FUNCTION_BLOCK Master_Axis
VAR_INPUT
	(*Linked_Axis		: AXIS_REF;*)
END_VAR
VAR_OUTPUT
END_VAR
VAR
	Linked_Axis		: AXIS_REF;
	// Motion Control Function Blocks
	Power				: MC_POWER;
	Pause				: MC_HALT;
	Reference_Drive		: MC_HOME;
	AbsoluteMotion		: MC_MOVEABSOLUTE;
	RelativeMotion		: MC_MOVERELATIVE;
	EmergencyStop		: MC_STOP;
	Axis_Jog			: MC_Jog;
	
	
	// Variables to operate functions of the axis
	PowerUp			: BOOL;
	Enable_Positive	: BOOL;
	Enable_Negative : BOOL;
	PowerOverride	: INT;
	PowerDown		: BOOL;
	
	Hault_Execute	: BOOL;
	HaultTrigger	: R_Trig;
	
	Lock_Axis		: BOOL;
	
	
	
	Home_Execute	: BOOL;
	HomeTrigger		: R_Trig;
	
	//MoveAbsolute Variables
	MoveAbsolute_Execute	: BOOL;
	MoveAbsoluteTrigger		: R_Trig;
	
	//MoveRelative Variabled
	MoveRelative_Execute	: BOOL;
	MoveRelativeTrigger		: R_Trig;
	
	
	//Structure that hold variables which are connected wirh the output side of the MC FBs
	Status 			: AxisFBStatus;
	
	// State Machine Variable for axis
	Machine_State			:	INT;
	Manual_State			:	INT;
	
	
	Jog_Positive	: BOOL;
	Jog_Negative	: BOOL;

END_VAR
VAR CONSTANT
	//Machine States 
	Machine_in_Automatic		:	INT := 1;
	Machine_in_Hand				:	INT	:= 2;
	Machine_in_Error			:	INT := 3;
	Machine_in_Undefined_State	:	INT := 4;

	//Axis States
	Manual_Move_Absolute	:	INT := 1;
	Manual_Move_Relative	:	INT := 2;
	Manual_Jog_Forward		:	INT := 3;
	Manual_Jog_Backward		:	INT := 4;
	Manual_Enable			:	INT := 5;
	Manual_Stop				: 	INT := 6;
	Manual_Lock				:	INT := 7;
	Manual_Home				:	INT := 8;
	Manual_Reset			:	INT := 9;
	
	
	
END_VAR

Power(Axis := Linked_Axis,
	   Enable:= Powerup,
	   Enable_Positive := Enable_Positive,
	   Enable_Negative := Enable_Negative,
	   Override := PowerOverride ,
	   BufferMode := ,
	   Options := ,
	   Status => Status.Power.Status,
	   Busy => Status.Power.Busy,
	   Active => Status.Power.Active,
	   Error => Status.Power.Error,
	   ErrorID => Status.Power.ErrorID);
	   
HaultTrigger(CLK := Hault_Execute);   
Pause(Axis := Linked_Axis,
	  Execute := Hault_Execute(*HaultTrigger.Q*),
	  Deceleration := ,
	  Jerk := ,
	  BufferMode := ,
	  Options := ,
	  Done => Status.Hault.Done ,
	  Busy => Status.Hault.Busy ,
	  Active => Status.Hault.Active,
	  CommandAborted => Status.Hault.CommandAborted,
	  Error => Status.Hault.Error,
	  ErrorID => Status.Hault.ErrorID);
	  
HomeTrigger(CLK := Home_Execute);
Reference_Drive(Axis := Linked_Axis,
	 Execute := HomeTrigger.Q,
	 Position := 0,
	 HomingMode := MC_Direct,
	 BufferMode := ,
	 Options := ,
	 bCalibrationCam := ,
	 Done => Status.Home.Done,
	 Busy => Status.Home.Busy,
	 Active => Status.Home.Active,
	 CommandAborted => Status.Home.CommandAborted,
	 Error => Status.Home.Error,
	 ErrorID => Status.Home.ErrorID);
	 
MoveAbsoluteTrigger(CLK:= MoveAbsolute_Execute);
AbsoluteMotion(Axis := Linked_Axis,
			 Execute := (*MoveAbsoluteTrigger.Q*)MoveAbsolute_Execute,
			 Position := 1500,
			 Velocity := 20,
			 Acceleration := 5,
			 Deceleration := 5,
			 Jerk := 5,
			 BufferMode := ,
			 Options := ,
			 Done => Status.MoveAbsolute.Done,
			 Busy => Status.MoveAbsolute.Busy,
			 Active => Status.MoveAbsolute.Active,
			 CommandAborted => Status.MoveAbsolute.CommandAborted,
			 Error => Status.MoveAbsolute.Error,
			 ErrorID => Status.MoveAbsolute.ErrorID);
			 
MoveRelativeTrigger(CLK := MoveRelative_Execute);
RelativeMotion(Axis := Linked_Axis,
			 Execute := MoveRelativeTrigger.Q,
			 Distance := 500,
			 Velocity := 10,
			 Acceleration := 1,
			 Deceleration := 1,
			 Jerk := 1,
		     BufferMode := ,
			 Options := ,
			 Done => Status.MoveRelative.Done,
			 Busy => Status.MoveRelative.Busy,
			 Active => Status.MoveRelative.Active,
			 CommandAborted => Status.MoveRelative.CommandAborted,
			 Error => Status.MoveRelative.Error,
			 ErrorID => Status.MoveRelative.ErrorID);			 

EmergencyStop(Axis := Linked_Axis,
			  Execute := Lock_Axis,
			  Deceleration := ,
			  Jerk := ,
			  Options := ,
			  Done => Status.Stop.Done,
			  Busy => Status.Stop.Busy,
			  Active => Status.Stop.Active,
			  CommandAborted => Status.Stop.CommandAborted,
			  Error => Status.Stop.Error,
			  ErrorID => Status.Stop.ErrorID);
			  
Axis_Jog(Axis := Linked_Axis,
		 JogForward := Jog_Positive,
		 JogBackwards := Jog_Negative,
		 Mode := ,
		 Position := MC_JOGMODE_CONTINOUS,
		 Velocity := ,
		 Acceleration := ,
		 Deceleration := ,
		 Jerk := ,
		 Done := ,
		 Busy := ,
		 Active := ,
		 CommandAborted := ,
		 Error := ,
		 ErrorID := );		  
		 
		 
CASE Machine_State OF
	
	Machine_in_Automatic :
	
	
	Machine_in_Hand:
		
			CASE Manual_State OF
			
				Manual_Enable:
	
				Manual_Move_Absolute:
	
				Manual_Move_Relative:
	
				Manual_Jog_Forward:
	
				Manual_Jog_Backward:
	
				Manual_Stop:
	
				Manual_Lock:
	
				Manual_Home:
	
				Manual_Reset:	
			
			END_CASE
		
	Machine_in_Error:
	
	
	Machine_in_Undefined_State:
	
	
END_CASE

PROPERTY Axis_State : BOOL
GET
END_GET
SET
END_SET
END_PROPERTY

METHOD Enable : BOOL
VAR_INPUT
END_VAR
PowerOverride := 100;
PowerUp := TRUE;
Enable_Positive := TRUE;
Enable_Negative := TRUE;

IF Status.Power.Status THEN
	Enable := TRUE;
END_IF
END_METHOD

METHOD Hault	: BOOL
VAR_INPUT
END_VAR
Hault_Execute := TRUE;

IF Status.Hault.Done THEN
	Hault := TRUE;
END_IF
END_METHOD

METHOD Home : BOOL
VAR_INPUT
END_VAR
Home_Execute := TRUE;

IF Status.Home.Done THEN
	Home_Execute := TRUE;
	Home := True;
END_IF
END_METHOD

METHOD MoveAbsolute : BOOL
VAR_INPUT
END_VAR
MoveAbsolute_Execute := TRUE;

IF Status.MoveAbsolute.Done THEN
	MoveAbsolute_Execute := FALSE;
	MoveAbsolute := TRUE;
END_IF
END_METHOD

METHOD MoveRelative : BOOL
VAR_INPUT
END_VAR
MoveRelative_Execute := TRUE;

IF Status.MoveRelative.Done THEN
	MoveRelative_Execute := FALSE;
	MoveRelative := TRUE;
END_IF
END_METHOD

METHOD Stop : BOOL
VAR_INPUT
END_VAR
Lock_Axis := TRUE;

IF Status.Stop.Done THEN
	Stop := TRUE;
END_IF
END_METHOD

END_FUNCTION_BLOCK

(* stored: Version 1.1.0.1, ProductVersion 3.1.4024.10
   POU Master_Axis: Id {667298e9-046b-4530-8e8f-220db46feb15}, SpecialFunc None
   Property Axis_State: Id {10fedc61-71d5-4610-bd9d-cec5bc6b893c}
   Get Get: Id {74911ec7-62b5-4dfd-8145-d7de79290190}
   Set Set: Id {8e6d4562-4d71-4a04-89bc-786582cc1f66}
   Method Enable: Id {d3be3a2f-5cc4-4162-bfd3-aadcfa398ae1}
   Method Hault: Id {bd6648fb-657d-4fdd-8fd7-45d948503f9c}
   Method Home: Id {4ab2e657-9053-4beb-a8ce-2a2b81376182}
   Method MoveAbsolute: Id {0ea4a38c-35e8-4c49-8844-b70ba6545c2f}
   Method MoveRelative: Id {a0368554-fdfb-46af-b2a7-920c35c033a5}
   Method Stop: Id {f38da706-b646-4e55-8636-403202df1783} *)
